FUNCTION_BLOCK LABELLING
  {SET_ATTRIBUTE(OpcUa, SERVICE)}
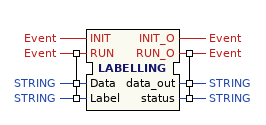
  EVENT_INPUT
    INIT;
    RUN WITH Data, Label; {SET_ATTRIBUTE(OpcUa, Method)}
  END_EVENT
  EVENT_OUTPUT
    INIT_O;
    RUN_O WITH data_out, status;
  END_EVENT
  VAR_INPUT
    Data : STRING; {SET_ATTRIBUTE(OpcUa, Variable.RUN)}
    Label : STRING; {SET_ATTRIBUTE(OpcUa, Variable.RUN)}
  END_VAR
  VAR_OUTPUT
    data_out : STRING; {SET_ATTRIBUTE(OpcUa, Variable.RUN)}
    status : STRING; {SET_ATTRIBUTE(OpcUa, Variable.RUN)}
  END_VAR
END_FUNCTION_BLOCK
